// TIA Portal V17 export
// export: Created 2024-09-02T12:50:35.2471616Z, ExportSetting WithDefaults, DisplayName Totally Integrated Automation Portal, DisplayVersion V17, DisplayName TIA Portal Openness, DisplayVersion V17, DisplayName TIA Portal Version Control Interface, DisplayVersion V17, DisplayName STEP 7 Professional, DisplayVersion V17, DisplayName STEP 7 Safety, DisplayVersion V17, DisplayName WinCC Professional, DisplayVersion V17
TYPE "TypeMobyGrunddaten_1"
// stored: IsFailsafeCompliant false
   STRUCT
      wt_kennung : Byte;   // 255 = WT ist bereits gelöscht / 255 = WT is already deleted
      palettenumlaufzaehler_h : Byte;   // H-Byte
      palettenumlaufzaehler_l : Byte;   // L-Byte / L byte
      paletten_nr_1000 : Char;   // 10^3
      paletten_nr_100 : Char;   // 10^2
      paletten_nr_10 : Char;   // 10^1
      paletten_nr_1 : Char;   // 10^0
      schlues_nr_res : Char;   // Schlüsselnummer Reserve / Button Number Reserve
      schlues_nr_1000 : Char;   // Schlüsselnummer 10^3 / Button Number 10^3
      schlues_nr_100 : Char;   // Schlüsselnummer 10^2 / Button Number 10^2
      schlues_nr_10 : Char;   // Schlüsselnummer 10^1 / Button Number 10^1
      schlues_nr_1 : Char;   // Schlüsselnummer 10^0 / Button Number 10^0
      res_12 : Byte;
      res_13 : Byte;
      losgroesse_10 : Byte;   // Losgröße 10^1 / Lot size 10^1
      losgroesse_1 : Byte;   // Losgröße 10^0 / Lot size 10^0
      Rest_10 : Byte;   // Rest 10^1
      Rest_1 : Byte;   // Rest 10^0
      res_18 : Byte;
      res_19 : Byte;
      res_20 : Byte;
      res_21 : Byte;
      kennung_01 : Char;   // Sonderkennung / Zielkennung / Special identifier / Destination identifier
      kennung_02 : Char;   // Sonderkennung / Zielkennung / Special identifier / Destination identifier
      Gruppe_10 : Char;   // Gruppe / Group
      Gruppe_1 : Char;   // Gruppe / Group
      res_26 : Byte;
      res_27 : Byte;
      Logistik_4 : Byte;   // Logistik / Logistic
      Logistik_3 : Byte;   // Logistik / Logistic
      Logistik_2 : Byte;   // Logistik / Logistic
      Logistik_1 : Byte;   // Logistik / Logistic
      res_32 : Byte;
      motor_nr_01 : Char;   // Laufende Nummer 10^5 / Serial number 10^5
      motor_nr_02 : Char;   // Laufende Nummer 10^4 / Serial number 10^4
      motor_nr_03 : Char;   // Laufende Nummer 10^3 / Serial number 10^3
      motor_nr_04 : Char;   // Laufende Nummer 10^2 / Serial number 10^2
      motor_nr_05 : Char;   // Laufende Nummer 10^1 / Serial number 10^1
      motor_nr_06 : Char;   // Laufende Nummer 10^0 / Serial number 10^0
      motor_nr_07 : Char;   // 1. Kennbuchstabe / 1. Code letter
      motor_nr_08 : Char;   // 2. Kennbuchstabe / 2. Code letter
      motor_nr_09 : Char;   // 3. Kennbuchstabe / 3. Code Letter
      res_42 : Byte;
      res_43 : Byte;
      datum_00 : Char;   // Tag 10^1
      datum_01 : Char;   // Tag 10^0
      datum_02 : Char;   // Monat 10^1 / Month 10^1
      datum_03 : Char;   // Monat 10^0 / Month 10^0
      datum_04 : Char;   // Jahr 10^1 / Year 10 ^ 1
      datum_05 : Char;   // Jahr 10^0 / Year 10 ^ 0
      datum_06 : Char;   // Stunde 10^1 / Hour 10^1
      datum_07 : Char;   // Stunde 10^0 / Hour 10^0
      datum_08 : Char;   // Minute 10^1
      datum_09 : Char;   // Minute 10^0
      res_54 : Byte;
      res_55 : Byte;
      res_56 : Byte;
      res_57 : Byte;
      res_58 : Byte;
      res_59 : Byte;
      folge_schlues_nr_res : Char;   // Schlüsselnummer Reserve / Button Number Reserve
      folge_schlues_nr_1000 : Char;   // Schlüsselnummer 10^3 / Button Number 10^3
      folge_schlues_nr_100 : Char;   // Schlüsselnummer 10^2 / Button Number 10^2
      folge_schlues_nr_10 : Char;   // Schlüsselnummer 10^1 / Button Number 10^1
      folge_schlues_nr_1 : Char;   // Schlüsselnummer 10^0 / Button Number 10^0
      PNR_Nr_01 : Char;   // Produktionsnummer / Production number
      PNR_Nr_02 : Char;   // Produktionsnummer / Production number
      PNR_Nr_03 : Char;   // Produktionsnummer / Production number
      PNR_Nr_04 : Char;   // Produktionsnummer / Production number
      PNR_Nr_05 : Char;   // Produktionsnummer / Production number
      PNR_Nr_06 : Char;   // Produktionsnummer / Production number
      PNR_Nr_07 : Char;   // Produktionsnummer / Production number
      PNR_Nr_08 : Char;   // Produktionsnummer / Production number
      PNR_Nr_09 : Char;   // Produktionsnummer / Production number
      PNR_Nr_10 : Char;   // Produktionsnummer / Production number
      res_75 : Byte;
      res_76 : Byte;
      res_77 : Byte;
      res_78 : Byte;
      res_79 : Byte;
      rumpf_paletten_nr_1000 : Char;   // Rumpf Palette-Nr. in Kalttest 10^3 / Hull pallet no. in cold test 10^3
      rumpf_paletten_nr_100 : Char;   // Rumpf Palette-Nr. in Kalttest 10^2 / Hull pallet no. in cold test 10^2
      rumpf_paletten_nr_10 : Char;   // Rumpf Palette-Nr. in Kalttest 10^1 / Hull pallet no. in cold test 10^1
      rumpf_paletten_nr_1 : Char;   // Rumpf Palette-Nr. in Kalttest 10^0 / Hull pallet no. in cold test 10^0
      reserve : Array[84..255] of Byte;
      wt_neutralisiert : Bool;   // WT neutralisiert / WT neutralized
      wt_manuell_nio : Bool;   // WT ohne weitere Bearbeitung zur nächsten E/A / WT to next I/O without further processing
      wt_leer : Bool;   // Leer WT / Empty WT
      motor_ohne_paergen : Bool;   // Motornummer nicht prägen / Do not emboss engine number
      staus_04 : Bool;   // feri
      staus_05 : Bool;   // feri
      staus_06 : Bool;   // feri
      staus_07 : Bool;   // feri
      loszaehler : Byte;   // wird bei jedem Start des Loses hochgezählt, um Änderung in der Schlüsselnummer / is incremented each time the lot is started in order to change the button number
      stapelzeiger_1 : Byte;   // Stapelzeiger auf Blockzeiger in Page 79 - 128 / Stack pointer to block pointer in Page 79 - 128
      stapelzeiger_2 : Byte;   // Stapelzeiger auf Blockzeiger in Page 79 - 128 / Stack pointer to block pointer in Page 79 - 128
      stapelzeigerEAS1_1 : Byte;   // Differenzzeiger für NA EAS1 / Differential pointer for NA EAS4
      stapelzeigerEAS1_2 : Byte;   // Differenzzeiger für NA EAS1 / Differential pointer for NA EAS4
      stapelzeigerEAS2_1 : Byte;   // Differenzzeiger für NA EAS1 / Differential pointer for NA EAS4
      stapelzeigerEAS2_2 : Byte;   // Differenzzeiger für NA EAS1 / Differential pointer for NA EAS4
      stapelzeigerEAS3_1 : Byte;   // Differenzzeiger für NA EAS1 / Differential pointer for NA EAS4
      stapelzeigerEAS3_2 : Byte;   // Differenzzeiger für NA EAS1 / Differential pointer for NA EAS4
      stapelzeigerEAS4_1 : Byte;   // Differenzzeiger für NA EAS1 / Differential pointer for NA EAS4
      stapelzeigerEAS4_2 : Byte;   // Differenzzeiger für NA EAS1 / Differential pointer for NA EAS4
      stapelzeigerEAS5_1 : Byte;   // Differenzzeiger für NA EAS1 / Differential pointer for NA EAS4
      stapelzeigerEAS5_2 : Byte;   // Differenzzeiger für NA EAS1 / Differential pointer for NA EAS4
      stapelzeigerEAS6_1 : Byte;   // Differenzzeiger für NA EAS1 / Differential pointer for NA EAS4
      stapelzeigerEAS6_2 : Byte;   // Differenzzeiger für NA EAS1 / Differential pointer for NA EAS4
      stapelzeigerEAS7_1 : Byte;   // Differenzzeiger für NA EAS1 / Differential pointer for NA EAS4
      stapelzeigerEAS7_2 : Byte;   // Differenzzeiger für NA EAS1 / Differential pointer for NA EAS4
      stapelzeigerEAS8_1 : Byte;   // Differenzzeiger für NA EAS1 / Differential pointer for NA EAS4
      stapelzeigerEAS8_2 : Byte;   // Differenzzeiger für NA EAS1 / Differential pointer for NA EAS4
      stapelzeigerEAS9_1 : Byte;   // Differenzzeiger für NA EAS1 / Differential pointer for NA EAS4
      stapelzeigerEAS9_2 : Byte;   // Differenzzeiger für NA EAS1 / Differential pointer for NA EAS4
      RES_278_bis_511 : Array[278..511] of Byte;   // Stationssonderdaten / Special ward data
   END_STRUCT;
END_TYPE
